TYPE DUT_SERVER_MODULE_INTERFACE_OUTPUT :
STRUCT
	///Free to use = TRUE, busy to use =FALSE
	Dummy: BOOL := TRUE;
	///Individual name of the module
	Name: STRING(80);
	///Identification number of module
	ID: UINT;
	///IP address
	IP: STRING(80);
	///Show if the module is in Standby or not
	Idle: BOOL;
	///Show if the module is connected
	Connected: BOOL;
	///Feedback with conection test input
	ConnectionTestOutput: BOOL;
	///Show if the system has error when=TRUE
	Error: BOOL;
	///Identification number of the error
	ErrorID: UINT;
	///Description of the error
	ErrorDescription: STRING(80);
	///Description of the current task
	CurrentTaskDescription: STRING(80);
	///Position of the output
	PositionOutput: LREAL;
	/// Bool value of the Sensor
	PositionSensor: BOOL;
	///Range of OUTPUT skills
	SkillOutput: DUT_SERVER_SKILLOUTPUTARRAY;
	///Range of state values
	StateValue: DUT_SERVER_STATEVALUEARRAY;
END_STRUCT
END_TYPE

(* stored: Version 1.1.0.1, ProductVersion 3.1.0.25
   DUT DUT_SERVER_MODULE_INTERFACE_OUTPUT: Id {09278e6c-87d3-4fa9-88d1-0b61e6d7c98d} *)
